TYPE EL3002_CHANNEL :
	STRUCT
		
	
	Status 	AT %I* : EL3002_DEV_STATUS;
	Value 	AT %I* : INT;
	
	
	END_STRUCT
END_TYPE

(* stored: Version 1.1.0.1
   DUT EL3002_CHANNEL: Id {72c41ae3-6521-41c2-b446-4199d1b594cf} *)
